PROGRAM MAIN


(*** CONTROLLERS: MAIN LOGIC MODULARIZED ***)

// Reactor temperature
ReactorTemperatureController(
						temperatureUpper := GVL_IO.reactorTemperatureUpper,
						temperatureLower := GVL_IO.reactorTemperatureLower,
						contactor => GVL_IO.reactorTemperatureContactor);

// Reactor level/pressure
ReactorLevelAndPressureController(
					serialCommData := SerialCommunicationController.SerialCommReadData,
					stop := SafetyController.stop,
					levelHigh := GVL_IO.reactorLevelHigh,
					slurryInletValve => GVL_IO.reactorInletValve,
					slurryOutletValve => GVL_IO.reactorOutletValve,
					extractiveOutletOnOffValve => GVL_IO.extractiveOutletOnOffValve,
					extractiveOutletControlValveClose => GVL_IO.extractiveOutletControlValveClose,
					extractiveOutletControlValveOpen => GVL_IO.extractiveOutletControlValveOpen);
					
// Data acquisition
DataAcquisitionController();

// Persistent data saving
VariablePersistenceController();

// Serial communication
SerialCommunicationController();

// Safety
SafetyController();

(*** VISUALIZATION BINDINGS: DATA TRANSFER FROM/TO UI ***)

// MainScreen in
MainScreenBindings(
				matlabValues := DataAcquisitionController.MatlabHmiValues,
				SerialCommReadData := SerialCommunicationController.SerialCommReadData,
				CalibrateDone := ReactorLevelAndPressureController.CalibrateDone,
				Stop :=  SafetyController.stop);
// MainScreen out
ReactorTemperatureController.autoControlSelected := MainScreenBindings.autoControlSelected;
ReactorTemperatureController.temperatureSetpoint := MainScreenBindings.temperatureSetpoint;
ReactorTemperatureController.manualControlPercentage := MainScreenBindings.temperaturePidManualControlPercentage;
DataAcquisitionController.MatlabBtn := MainScreenBindings.matlabBtn;
GVL_OPC.OPC_ProgramNamePrefix := MainScreenBindings.programNamePrefix;
ReactorLevelAndPressureController.StartAutomaticExtraction := MainScreenBindings.startAutomaticExtraction;
SafetyController.buttonPressed := MainScreenBindings.estopButtonPressed;
SafetyController.resetPressed := MainScreenBindings.estopResetPressed;
SerialCommunicationController.SerialCommSetpoints := MainScreenBindings.serialCommSetpoints;
	
//ProcessView in			
ProcessViewBindings(
				reactorOutletValve := GVL_IO.reactorOutletValve,
				reactorInletValve := GVL_IO.reactorInletValve,
				lowerTemperature := ReactorTemperatureController.lowerTemperature,
				upperTemperature := ReactorTemperatureController.upperTemperature,
				reactorTemperatureContactor := GVL_IO.reactorTemperatureContactor,
				reactorLevelHigh := GVL_IO.reactorLevelHigh,
				reactorLevelLow := GVL_IO.reactorLevelLow,
				iPressureScaledValue := ReactorLevelAndPressureController.iPressureScaledValue,
				SerialCommReadData := SerialCommunicationController.SerialCommReadData,
				ExtractiveOnOffValveValues := ReactorLevelAndPressureController.ExtractiveOnOffValveValues,
				CalibrateDone := ReactorLevelAndPressureController.CalibrateDone,
				ControlValveOpening := ReactorLevelAndPressureController.ControlValveOpening,
				automaticExtractionState := ReactorLevelAndPressureController.automaticExtractionState,
				stop := SafetyController.stop);
// ProcessView out
ReactorTemperatureController.temperatureContactorCommand := ProcessViewBindings.temperatureContactorCommand;
ReactorLevelAndPressureController.SlurryInValveCommand := ProcessViewBindings.SlurryInValveCommand;
ReactorLevelAndPressureController.PressureIntervals := ProcessViewBindings.PressureIntervals;
ReactorLevelAndPressureController.SlurryOutValveCommand := ProcessViewBindings.SlurryOutValveCommand;
ReactorLevelAndPressureController.ExtractiveOutOnOffValveCommand := ProcessViewBindings.ExtractiveOutOnOffValveCommand;
ReactorLevelAndPressureController.ExtractiveControlValveCommands := ProcessViewBindings.ExtractiveControlValveCommands;
	
// ParameterView in			
ParameterViewBindings();
// ParameterView out
ReactorTemperatureController.pidControllerParameters := ParameterViewBindings.reactorTemperaturePidParameters;
ReactorLevelAndPressureController.AutomaticExtractionParameters := ParameterViewBindings.autoExtractionParameters;
ReactorLevelAndPressureController.PressureIntervals := ParameterViewBindings.pressureIntervals;
ReactorLevelAndPressureController.ExtractiveControlValveParameters := ParameterViewBindings.extractionValveParameters;

END_PROGRAM

(* stored: Version 1.1.0.1, ProductVersion 3.1.4024.9
   POU MAIN: Id {dec5b1ca-8e16-4f49-8efb-57a750654862}, SpecialFunc None *)
